{attribute 'qualified_only'}
{attribute 'strict'}
{attribute 'to_string'}
TYPE E_nozzleState :
(
	disabled := 0,
	standby := 1,
	refuelling := 2
)DINT;
END_TYPE

(* stored: Version 1.1.0.1
   DUT E_nozzleState: Id {817bb791-e2e7-40ee-a522-a92d4dfc831d} *)
